# EPICS autosave request: softGlueApp/Db/MUX2_settings.req
$(P)$(H)MUX2-$(N)_desc
$(P)$(H)MUX2-$(N)_IN0_Signal
$(P)$(H)MUX2-$(N)_IN1_Signal
$(P)$(H)MUX2-$(N)_OUT_Signal
$(P)$(H)MUX2-$(N)_SEL_Signal
